(* PLC project average, Dassault Systèmes ControlBuild 2024x *)
(* stored: creationDateTime 2023-10-03T11:13:27-01:00 *)

(* This module returns a real. This real corresponds to the average value of two real inputs. *)
FUNCTION_BLOCK equipment_library.average
  VAR_INPUT
    input1 : REAL := 0.0;
    input2 : REAL := 0.0;
  END_VAR
  VAR_OUTPUT
    result : REAL := 0.0;
  END_VAR
  VAR
    d_average : BOOL := false;
    v_d_average : REAL := 0.0;
  END_VAR


ACTION C_source_code:
/* ----------------------------------------------------------------	*/
/* Type : Model of Operative Behaviour					*/
/* Category :  Toolbox							*/
/* Author : Dassault Systemes						*/
/* Update date : June 2018						*/
/* ----------------------------------------------------------------	*/
/* This module returns a real. 						*/
/* This real corresponds to the average value of two real inputs.	*/
/* ----------------------------------------------------------------	*/

if (d_average) result = v_d_average;	 /* presetting of the value */
else result = ( input1 + input2 ) / 2.0;	/* result */
END_ACTION
END_FUNCTION_BLOCK
